// Mitsubishi GX Works2 project: 分拣项目   PLC: FX3U/FX3UC

PROGRAM MAIN  // 主程序
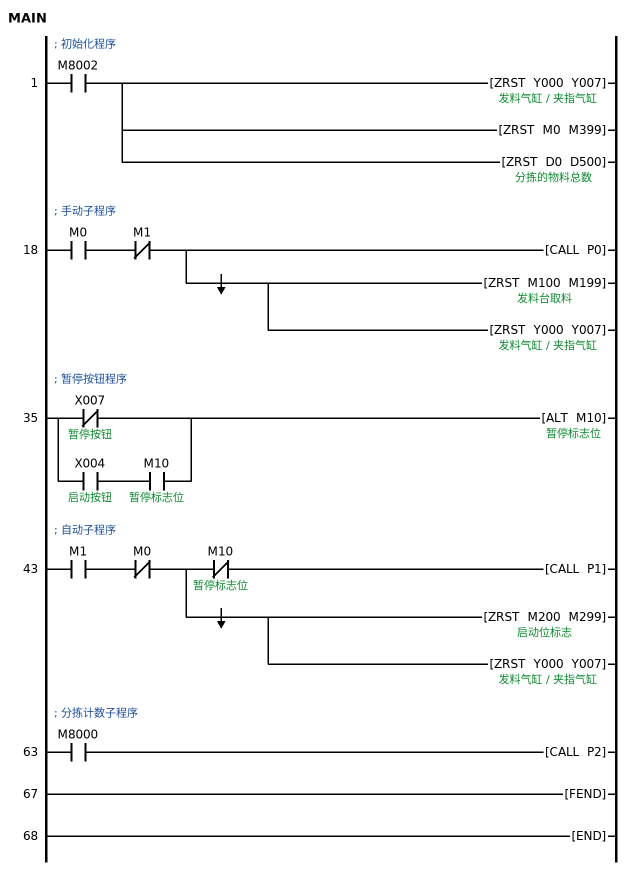
; 初始化程序
1     LD      M8002
      ZRST    Y000 Y007  ; 发料气缸 / 夹指气缸
      ZRST    M0 M399
      ZRST    D0 D500  ; 分拣的物料总数
; 手动子程序
18    LD      M0
      ANI     M1
      CALL    P0
      MEF
      ZRST    M100 M199  ; 发料台取料
      ZRST    Y000 Y007
; 暂停按钮程序
35    LDI     X007  ; 暂停按钮
      LD      X004  ; 启动按钮
      AND     M10  ; 暂停标志位
      ORB
      ALT     M10
; 自动子程序
43    LD      M1
      ANI     M0
      MPS
      ANI     M10  ; 暂停标志位
      CALL    P1
      MPP
      MEF
      ZRST    M200 M299  ; 启动位标志
      ZRST    Y000 Y007
; 分拣计数子程序
63    LD      M8000
      CALL    P2
67    FEND
68    END
END_PROGRAM

PROGRAM MAIN1  // 手动子程序
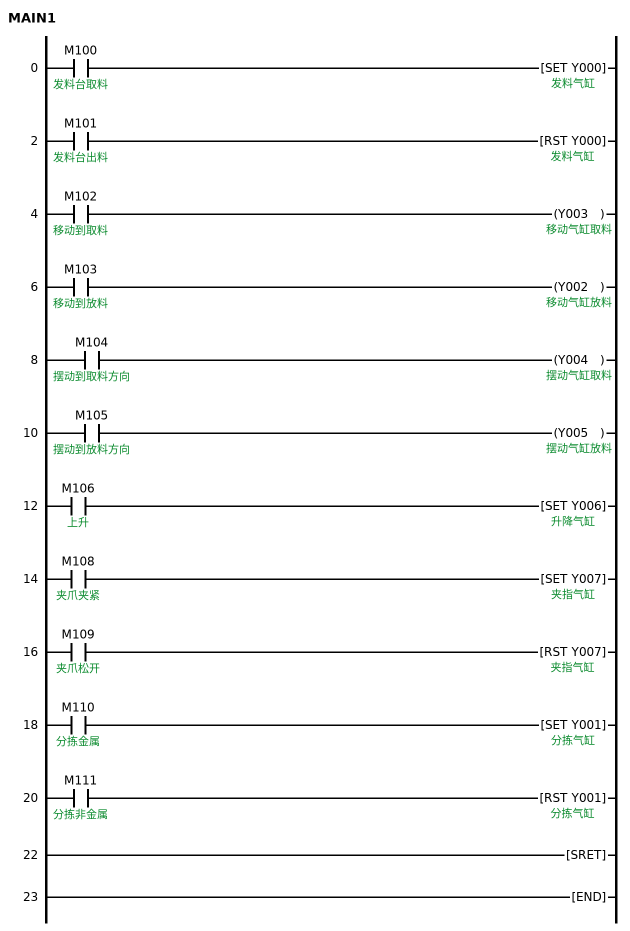
0     LD      M100  ; 发料台取料
      SET     Y000  ; 发料气缸
2     LD      M101  ; 发料台出料
      RST     Y000  ; 发料气缸
4     LD      M102  ; 移动到取料
      OUT     Y003  ; 移动气缸取料
6     LD      M103  ; 移动到放料
      OUT     Y002  ; 移动气缸放料
8     LD      M104  ; 摆动到取料方向
      OUT     Y004  ; 摆动气缸取料
10    LD      M105  ; 摆动到放料方向
      OUT     Y005  ; 摆动气缸放料
12    LD      M106  ; 上升
      SET     Y006  ; 升降气缸
14    LD      M108  ; 夹爪夹紧
      SET     Y007  ; 夹指气缸
16    LD      M109  ; 夹爪松开
      RST     Y007  ; 夹指气缸
18    LD      M110  ; 分拣金属
      SET     Y001  ; 分拣气缸
20    LD      M111  ; 分拣非金属
      RST     Y001  ; 分拣气缸
22    SRET
23    END
END_PROGRAM

PROGRAM MAIN2  // 自动子程序
      P1
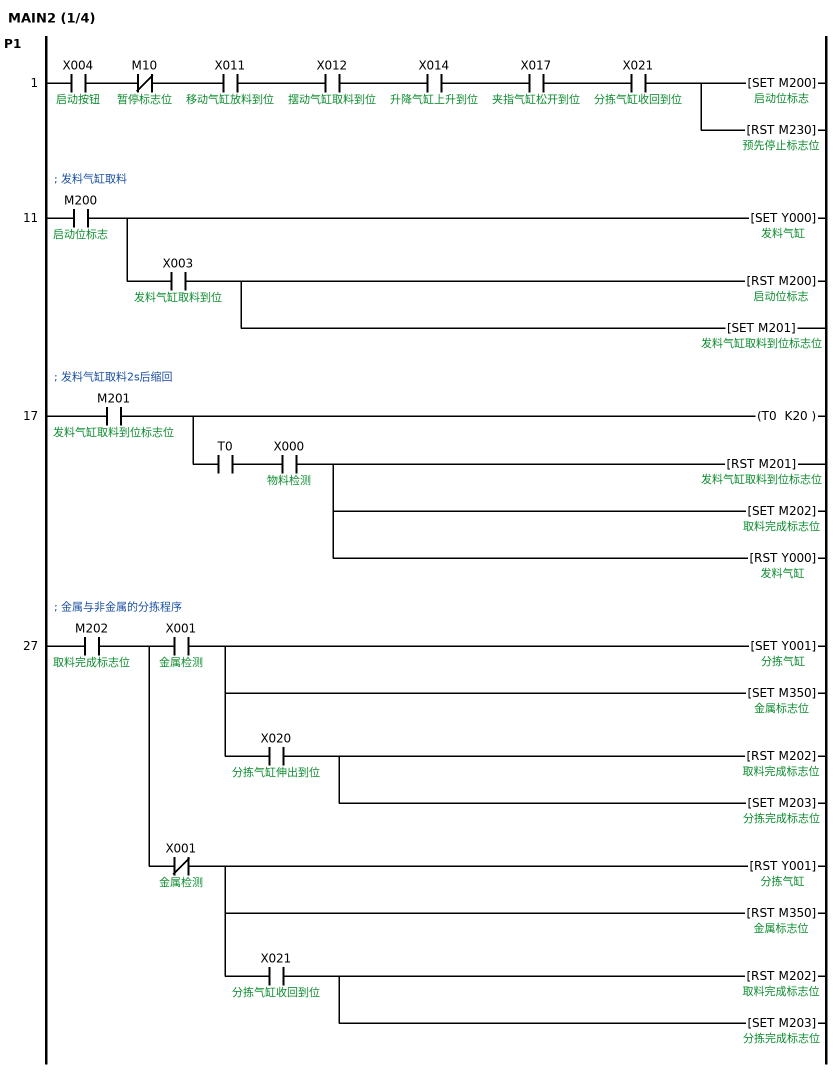
1     LD      X004  ; 启动按钮
      ANI     M10  ; 暂停标志位
      AND     X011  ; 移动气缸放料到位
      AND     X012  ; 摆动气缸取料到位
      AND     X014  ; 升降气缸上升到位
      AND     X017  ; 夹指气缸松开到位
      AND     X021  ; 分拣气缸收回到位
      SET     M200  ; 启动位标志
      RST     M230  ; 预先停止标志位
; 发料气缸取料
11    LD      M200  ; 启动位标志
      SET     Y000  ; 发料气缸
      AND     X003  ; 发料气缸取料到位
      RST     M200  ; 启动位标志
      SET     M201  ; 发料气缸取料到位标志位
; 发料气缸取料2s后缩回
17    LD      M201  ; 发料气缸取料到位标志位
      OUT     T0 K20
      AND     T0
      AND     X000  ; 物料检测
      RST     M201  ; 发料气缸取料到位标志位
      SET     M202  ; 取料完成标志位
      RST     Y000  ; 发料气缸
; 金属与非金属的分拣程序
27    LD      M202  ; 取料完成标志位
      MPS
      AND     X001  ; 金属检测
      SET     Y001  ; 分拣气缸
      SET     M350  ; 金属标志位
      AND     X020  ; 分拣气缸伸出到位
      RST     M202  ; 取料完成标志位
      SET     M203  ; 分拣完成标志位
      MPP
      ANI     X001  ; 金属检测
      RST     Y001  ; 分拣气缸
      RST     M350  ; 金属标志位
      AND     X021  ; 分拣气缸收回到位
      RST     M202  ; 取料完成标志位
      SET     M203  ; 分拣完成标志位
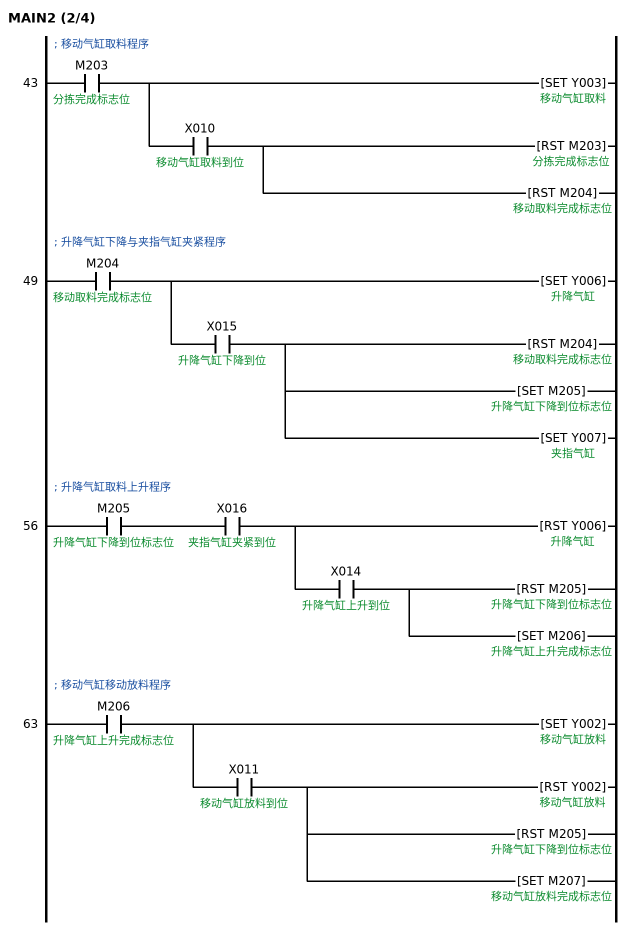
; 移动气缸取料程序
43    LD      M203  ; 分拣完成标志位
      SET     Y003  ; 移动气缸取料
      AND     X010  ; 移动气缸取料到位
      RST     M203  ; 分拣完成标志位
      RST     M204  ; 移动取料完成标志位
; 升降气缸下降与夹指气缸夹紧程序
49    LD      M204  ; 移动取料完成标志位
      SET     Y006  ; 升降气缸
      AND     X015  ; 升降气缸下降到位
      RST     M204  ; 移动取料完成标志位
      SET     M205  ; 升降气缸下降到位标志位
      SET     Y007  ; 夹指气缸
; 升降气缸取料上升程序
56    LD      M205  ; 升降气缸下降到位标志位
      AND     X016  ; 夹指气缸夹紧到位
      RST     Y006  ; 升降气缸
      AND     X014  ; 升降气缸上升到位
      RST     M205  ; 升降气缸下降到位标志位
      SET     M206  ; 升降气缸上升完成标志位
; 移动气缸移动放料程序
63    LD      M206  ; 升降气缸上升完成标志位
      SET     Y002  ; 移动气缸放料
      AND     X011  ; 移动气缸放料到位
      RST     Y002  ; 移动气缸放料
      RST     M205  ; 升降气缸下降到位标志位
      SET     M207  ; 移动气缸放料完成标志位
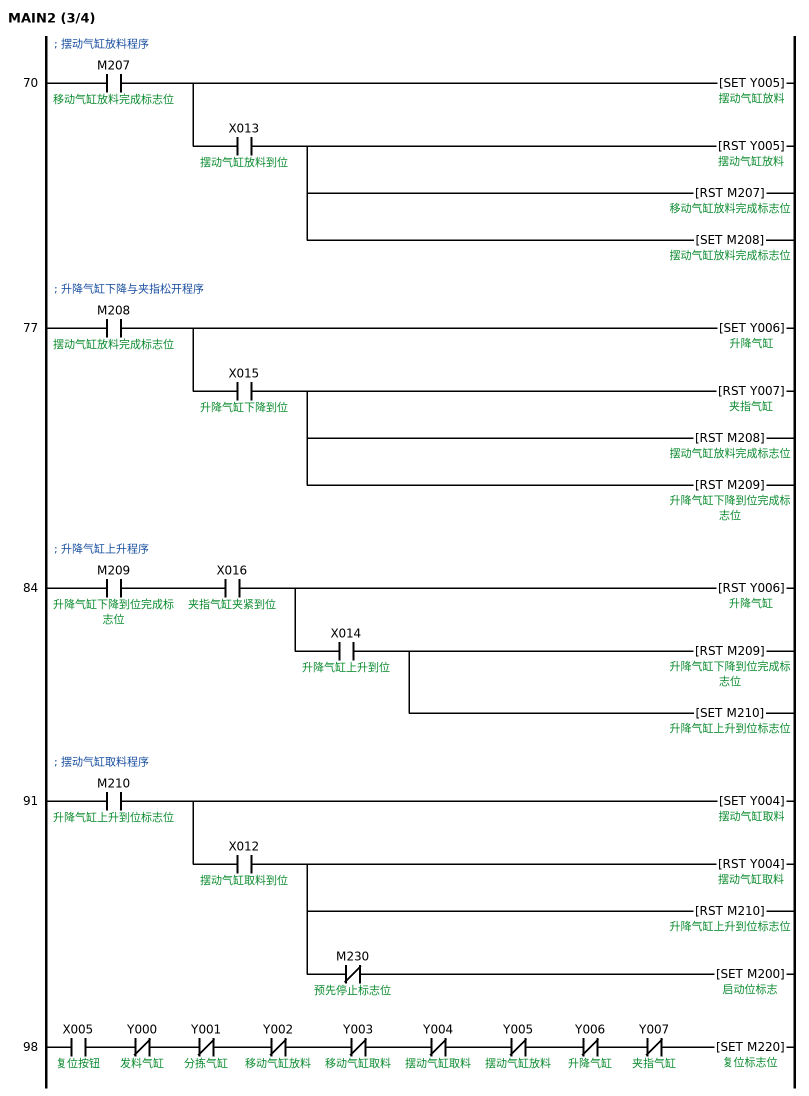
; 摆动气缸放料程序
70    LD      M207  ; 移动气缸放料完成标志位
      SET     Y005  ; 摆动气缸放料
      AND     X013  ; 摆动气缸放料到位
      RST     Y005  ; 摆动气缸放料
      RST     M207  ; 移动气缸放料完成标志位
      SET     M208  ; 摆动气缸放料完成标志位
; 升降气缸下降与夹指松开程序
77    LD      M208  ; 摆动气缸放料完成标志位
      SET     Y006  ; 升降气缸
      AND     X015  ; 升降气缸下降到位
      RST     Y007  ; 夹指气缸
      RST     M208  ; 摆动气缸放料完成标志位
      RST     M209  ; 升降气缸下降到位完成标志位
; 升降气缸上升程序
84    LD      M209  ; 升降气缸下降到位完成标志位
      AND     X016  ; 夹指气缸夹紧到位
      RST     Y006  ; 升降气缸
      AND     X014  ; 升降气缸上升到位
      RST     M209  ; 升降气缸下降到位完成标志位
      SET     M210  ; 升降气缸上升到位标志位
; 摆动气缸取料程序
91    LD      M210  ; 升降气缸上升到位标志位
      SET     Y004  ; 摆动气缸取料
      AND     X012  ; 摆动气缸取料到位
      RST     Y004  ; 摆动气缸取料
      RST     M210  ; 升降气缸上升到位标志位
      ANI     M230  ; 预先停止标志位
      SET     M200  ; 启动位标志
98    LD      X005  ; 复位按钮
      ANI     Y000  ; 发料气缸
      ANI     Y001  ; 分拣气缸
      ANI     Y002  ; 移动气缸放料
      ANI     Y003  ; 移动气缸取料
      ANI     Y004  ; 摆动气缸取料
      ANI     Y005  ; 摆动气缸放料
      ANI     Y006  ; 升降气缸
      ANI     Y007  ; 夹指气缸
      SET     M220  ; 复位标志位
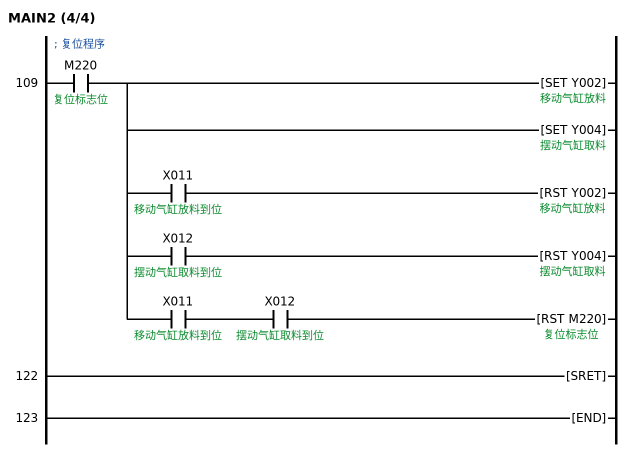
; 复位程序
109   LD      M220  ; 复位标志位
      SET     Y002  ; 移动气缸放料
      SET     Y004  ; 摆动气缸取料
      MPS
      AND     X011  ; 移动气缸放料到位
      RST     Y002  ; 移动气缸放料
      MRD
      AND     X012  ; 摆动气缸取料到位
      RST     Y004  ; 摆动气缸取料
      MPP
      AND     X011  ; 移动气缸放料到位
      AND     X012  ; 摆动气缸取料到位
      RST     M220  ; 复位标志位
122   SRET
123   END
END_PROGRAM

PROGRAM MAIN3  // 分拣计数子程序
      P2
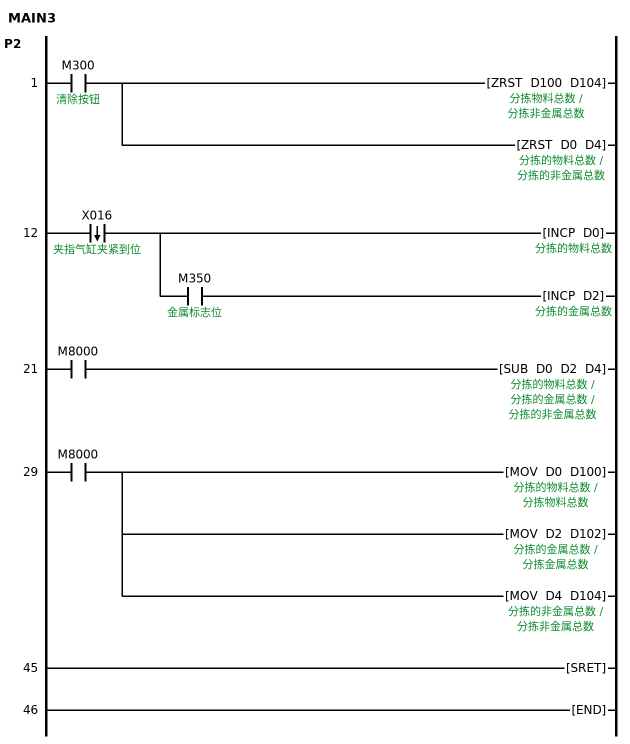
1     LD      M300  ; 清除按钮
      ZRST    D100 D104  ; 分拣物料总数 / 分拣非金属总数
      ZRST    D0 D4  ; 分拣的物料总数 / 分拣的非金属总数
12    LDF     X016  ; 夹指气缸夹紧到位
      INCP    D0
      AND     M350  ; 金属标志位
      INCP    D2  ; 分拣的金属总数
21    LD      M8000
      SUB     D0 D2 D4
29    LD      M8000
      MOV     D0 D100
      MOV     D2 D102  ; 分拣金属总数
      MOV     D4 D104
45    SRET
46    END
END_PROGRAM

// device comments not shown above
X002  ; 发料气放料到位
X006  ; 预停按钮
M107  ; 下降
